FUNCTION_BLOCK FB_TelescopeIdleState EXTENDS FB_TelescopeState
VAR_INPUT
END_VAR
VAR_OUTPUT
END_VAR
VAR
	pMachine : POINTER TO FB_TelescopeMachine;
END_VAR

METHOD FB_init : BOOL
VAR_INPUT
	bInitRetains : BOOL; // if TRUE, the retain variables are initialized (warm start / cold start)
	bInCopyCode : BOOL;  // if TRUE, the instance afterwards gets moved into the copy code (online change)
	pMachine : POINTER TO FB_TelescopeMachine;
END_VAR
THIS^.pMachine := pMachine;
END_METHOD

METHOD Park : BOOL
VAR_INPUT
END_VAR
END_METHOD

METHOD Slew : BOOL
VAR_INPUT
	fAzimuth	: LREAL;
	fAltitude	: LREAL;
END_VAR
END_METHOD

METHOD Track : BOOL
VAR_INPUT
	fRightAscension	: LREAL;
	fDeclination	: LREAL;
END_VAR
END_METHOD

END_FUNCTION_BLOCK

(* stored: Version 1.1.0.1, ProductVersion 3.1.4024.15
   POU FB_TelescopeIdleState: Id {97cb9578-1d5b-4b37-b757-b2f2bee04a18}, SpecialFunc None
   Method FB_init: Id {c6b8f45b-6fc8-481b-aaa5-568f5d8889b1}
   Method Park: Id {b4c875aa-42a3-40df-abd5-00dd16ea6370}
   Method Slew: Id {e8a6077b-8fe1-44d4-9a66-ac64e9f8ab2e}
   Method Track: Id {db24f220-0cc3-4d50-b558-3436eb190c49} *)
